// TIA Portal project "P7_P3_sim" (V14)

(* hardware
DEVICE "S7-1200 station_1"  S7-1200 Station
   slot 0: "Rack_0"  S7-1200 Rack  Rack  V1.0
   slot 1: "PLC_1"  CPU 1214C DC/DC/DC  6ES7 214-1AG40-0XB0  V4.2
*)

// ===== PLC "PLC_1"  CPU 1214C DC/DC/DC =====

VAR_GLOBAL   // PLC tag table "Default tag table"
   ""PM"" AT %I0.0 : Bool;
   ""PP"" AT %I0.1 : Bool;
   ""LUZ_AMARILLA"" AT %Q0.0 : Bool;
   ""LUZ_ROJA"" AT %Q0.1 : Bool;
   ""LUZ_VERDE"" AT %Q0.2 : Bool;
END_VAR